SUBAPPLICATION logiBUS_AI_Calibrated_Subscribe_VT_3P_OPC (* 3-Punkt-Pendant zu logiBUS_AI_Calibrated_Subscribe_VT_OPC (fuer Sensoren mit Mittelstellung, z.B. Neigungswinkel Hangausgleich B14): Remote-Subscribe eines bereits kalibrierten physikalischen Werts (M2M, von der Sensor-Station) -> VT-Anzeige + lokaler Re-Publish. Die physischen VT-Elemente bleiben hier (dort wo die VT ist): C_MIN/C_MID/C_MAX-Tasten rufen per CLIENT_0 direkt die ID_MIN_METHOD/ID_MID_TRIGGER_METHOD/ID_MAX_METHOD auf der Sensor-Station auf (logiBUS_AI_Calibrate_3P_IDA_OPC) - echter Event-zu-Event-Methodenaufruf, kein Toggle/Publish/Subscribe-Umweg (siehe OPC_UA_VERNETZUNG.md Punkt 14). MIN_REF/MID_REF/MAX_REF-Referenzwert-Eingabefelder bleiben bewusst aussen vor dieser SubApp (siehe Schnitthoehe_Winkel_Zero/SpanInput-Vorbild in Inputs_STG1.SUB) - eigene NumericValue_TO_CLIENT_1_0_OPC-Instanzen je Aufrufer. *)
  (* Standard: 61499-2; Description: Copyright (c) 2026 Meisterschulen am Ostbahnhof This program and the accompanying materials are made available under the terms of the Eclipse Public License 2.0 which is available at https://www.eclipse.org/legal/epl-2.0/ SPDX-License-Identifier: EPL-2.0 *)
  (* Version 1.1, 2026-09-26, Franz Höpfinger, Meisterschulen am Ostbahnhof, Neuer Plug CAL_OUT (AR) ergaenzt, analog logiBUS_AI_Calibrated_Subscribe_VT_OPC.CAL_OUT - Franz: 'ist das ein extra forwarding noetig? Fuer die CAL-Maske brauchen wir den kalibrierten Wert ohnehin schon' - genau dieser Plug spiegelt den bereits remote abonnierten Wert als lokalen AR-Plug fuer weitere Konsumenten auf STG1 (z.B. Fahrwerk_Mittelpunkt_Anzeige fuer Bargraph/Status-Center), kein zusaetzliches Self-Subscribe noetig. *)
  (* Version 1.0, 2026-09-26, Franz Höpfinger, Meisterschulen am Ostbahnhof, initial implementation - 3-Punkt-Pendant zu logiBUS_AI_Calibrated_Subscribe_VT_OPC v1.8, fuer Hangausgleich-Winkel B14 (Kalibrierung zieht von STG1 nach STG3 um). Franz: 'Klar B. Alles mit call method'. *)
  PACKAGE MyLib::sys;
  IMPORT isobus::UT::Q::const::IDs::ID_NULL;
  IMPORT isobus::UT::io::Button::ButtonActivationCode::BT_PRESSED_LATCHED;
  IMPORT logiBUS::utils::conversion::phys::NumericObjectPool_S;
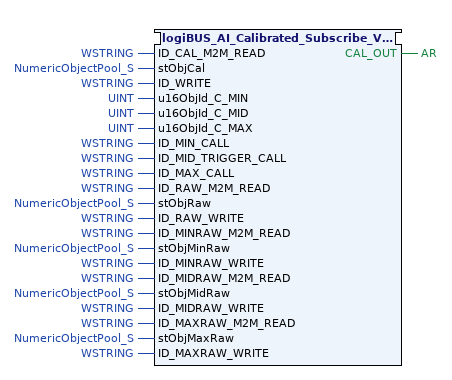
  VAR_INPUT
    ID_CAL_M2M_READ : WSTRING; (* Remote-Subscribe-Adresse des bereits kalibrierten physikalischen Werts (REAL) - Gegenstueck zu ID_CAL_WRITE auf der Sensor-Station (logiBUS_AI_Calibrate_3P_IDA_OPC) *)
    stObjCal : logiBUS::utils::conversion::phys::NumericObjectPool_S := (u16ObjId := ID_NULL, r32Scale := 1.0, i32Offset := 0, u8Decimals := 1); (* Object ID + Scale/Offset/Decimals CNumberVariable (kalibrierter Wert) *)
    ID_WRITE : WSTRING; (* Lokale Re-Publish-Adresse (REAL, ACTION=PUBLISH) fuer weitere lokale Konsumenten auf dieser Station *)
    u16ObjId_C_MIN : UINT := ID_NULL; (* Object ID Taste 'C_MIN' - physisch hier auf der VT *)
    u16ObjId_C_MID : UINT := ID_NULL; (* Object ID Taste 'C_MID' - physisch hier auf der VT *)
    u16ObjId_C_MAX : UINT := ID_NULL; (* Object ID Taste 'C_MAX' - physisch hier auf der VT *)
    ID_MIN_CALL : WSTRING; (* Remote-Methodenadresse (ACTION=CALL_METHOD) fuer den C_MIN-Trigger - ruft ID_MIN_METHOD direkt auf der Sensor-Station auf (logiBUS_AI_Calibrate_3P_IDA_OPC) *)
    ID_MID_TRIGGER_CALL : WSTRING; (* Remote-Methodenadresse (ACTION=CALL_METHOD) fuer den C_MID-Trigger - ruft ID_MID_TRIGGER_METHOD direkt auf der Sensor-Station auf *)
    ID_MAX_CALL : WSTRING; (* Remote-Methodenadresse (ACTION=CALL_METHOD) fuer den C_MAX-Trigger - ruft ID_MAX_METHOD direkt auf der Sensor-Station auf *)
    ID_RAW_M2M_READ : WSTRING; (* Remote-Subscribe-Adresse des unkalibrierten Rohwerts (DWORD 0-4095, reine Diagnose-Anzeige) - Gegenstueck zu ID_RAW_WRITE auf der Sensor-Station *)
    stObjRaw : logiBUS::utils::conversion::phys::NumericObjectPool_S := (u16ObjId := ID_NULL, r32Scale := 1.0, i32Offset := 0, u8Decimals := 0); (* Object ID + Scale/Offset/Decimals CNumberVariable (Rohwert-Anzeige) *)
    ID_RAW_WRITE : WSTRING; (* Lokale Re-Publish-Adresse (DWORD, ACTION=PUBLISH) fuer weitere lokale Konsumenten auf dieser Station *)
    ID_MINRAW_M2M_READ : WSTRING; (* Remote-Subscribe-Adresse des Rohwerts am MIN-Kalibrierpunkt (reine Diagnose-Anzeige) - Gegenstueck zu ID_MIN_RAW_WRITE auf der Sensor-Station *)
    stObjMinRaw : logiBUS::utils::conversion::phys::NumericObjectPool_S := (u16ObjId := ID_NULL, r32Scale := 1.0, i32Offset := 0, u8Decimals := 0); (* Object ID + Scale/Offset/Decimals CNumberVariable (Rohwert-Anzeige am MIN-Kalibrierpunkt) *)
    ID_MINRAW_WRITE : WSTRING; (* Lokale Re-Publish-Adresse (DWORD, ACTION=PUBLISH) fuer weitere lokale Konsumenten auf dieser Station *)
    ID_MIDRAW_M2M_READ : WSTRING; (* Remote-Subscribe-Adresse des Rohwerts am MID-Kalibrierpunkt (reine Diagnose-Anzeige) - Gegenstueck zu ID_MID_RAW_WRITE auf der Sensor-Station *)
    stObjMidRaw : logiBUS::utils::conversion::phys::NumericObjectPool_S := (u16ObjId := ID_NULL, r32Scale := 1.0, i32Offset := 0, u8Decimals := 0); (* Object ID + Scale/Offset/Decimals CNumberVariable (Rohwert-Anzeige am MID-Kalibrierpunkt) *)
    ID_MIDRAW_WRITE : WSTRING; (* Lokale Re-Publish-Adresse (DWORD, ACTION=PUBLISH) fuer weitere lokale Konsumenten auf dieser Station *)
    ID_MAXRAW_M2M_READ : WSTRING; (* Remote-Subscribe-Adresse des Rohwerts am MAX-Kalibrierpunkt (reine Diagnose-Anzeige) - Gegenstueck zu ID_MAX_RAW_WRITE auf der Sensor-Station *)
    stObjMaxRaw : logiBUS::utils::conversion::phys::NumericObjectPool_S := (u16ObjId := ID_NULL, r32Scale := 1.0, i32Offset := 0, u8Decimals := 0); (* Object ID + Scale/Offset/Decimals CNumberVariable (Rohwert-Anzeige am MAX-Kalibrierpunkt) *)
    ID_MAXRAW_WRITE : WSTRING; (* Lokale Re-Publish-Adresse (DWORD, ACTION=PUBLISH) fuer weitere lokale Konsumenten auf dieser Station *)
  END_VAR
  PLUGS
    CAL_OUT : adapter::types::unidirectional::AR; (* Nur-Lese-Spiegel des kalibrierten Werts (= ValueDisplay.VALUE_OUT) fuer weitere lokale Konsumenten auf dieser Station, statt eigenem OPC-UA-Self-Subscribe *)
  END_PLUGS
  SUBAPPS
    ValueDisplay : MyLib::sys::AR_M2M_Subscribe_TO_Q_Publish_OPC;
    TriggerMIN : MyLib::sys::Button_CLIENT_Method_IE(InputEvent := BT_PRESSED_LATCHED);
    TriggerMID : MyLib::sys::Button_CLIENT_Method_IE(InputEvent := BT_PRESSED_LATCHED);
    TriggerMAX : MyLib::sys::Button_CLIENT_Method_IE(InputEvent := BT_PRESSED_LATCHED);
    RawDisplay : MyLib::sys::AR_M2M_Subscribe_TO_Q_Publish_OPC;
    MinRawDisplay : MyLib::sys::AR_M2M_Subscribe_TO_Q_Publish_OPC;
    MidRawDisplay : MyLib::sys::AR_M2M_Subscribe_TO_Q_Publish_OPC;
    MaxRawDisplay : MyLib::sys::AR_M2M_Subscribe_TO_Q_Publish_OPC;
  END_SUBAPPS
  DATA_CONNECTIONS
    ID_CAL_M2M_READ TO ValueDisplay.ID_M2M_READ;
    stObjCal TO ValueDisplay.stObj;
    ID_WRITE TO ValueDisplay.ID_WRITE;
    u16ObjId_C_MIN TO TriggerMIN.u16ObjId;
    u16ObjId_C_MID TO TriggerMID.u16ObjId;
    u16ObjId_C_MAX TO TriggerMAX.u16ObjId;
    ID_MIN_CALL TO TriggerMIN.ID_CALL;
    ID_MID_TRIGGER_CALL TO TriggerMID.ID_CALL;
    ID_MAX_CALL TO TriggerMAX.ID_CALL;
    ID_RAW_M2M_READ TO RawDisplay.ID_M2M_READ;
    stObjRaw TO RawDisplay.stObj;
    ID_RAW_WRITE TO RawDisplay.ID_WRITE;
    ID_MINRAW_M2M_READ TO MinRawDisplay.ID_M2M_READ;
    stObjMinRaw TO MinRawDisplay.stObj;
    ID_MINRAW_WRITE TO MinRawDisplay.ID_WRITE;
    ID_MIDRAW_M2M_READ TO MidRawDisplay.ID_M2M_READ;
    stObjMidRaw TO MidRawDisplay.stObj;
    ID_MIDRAW_WRITE TO MidRawDisplay.ID_WRITE;
    ID_MAXRAW_M2M_READ TO MaxRawDisplay.ID_M2M_READ;
    stObjMaxRaw TO MaxRawDisplay.stObj;
    ID_MAXRAW_WRITE TO MaxRawDisplay.ID_WRITE;
  END_CONNECTIONS
  ADAPTER_CONNECTIONS
    ValueDisplay.VALUE_OUT TO CAL_OUT;
  END_CONNECTIONS
END_SUBAPPLICATION
